(*
Standard way to set up time events in a system. might make an interface
*)
FUNCTION_BLOCK ABSTRACT FB_TimeEvents
VAR_INPUT
END_VAR
VAR_OUTPUT
END_VAR
VAR
END_VAR

END_FUNCTION_BLOCK

(* stored: Version 1.1.0.1, ProductVersion 3.1.4024.12
   POU FB_TimeEvents: Id {67b3410e-360f-4a3a-95e0-d47352cef831}, SpecialFunc None *)
